Fanuc TP program (LS listing): HOME.LS

/PROG  HOME
/ATTR
OWNER		= MNEDITOR;
COMMENT		= "RobotSafePos";
PROG_SIZE	= 174;
CREATE		= DATE 26-08-17  TIME 11:20:48;
MODIFIED	= DATE 26-08-17  TIME 11:22:56;
FILE_NAME	= ;
VERSION		= 0;
LINE_COUNT	= 4;
MEMORY_SIZE	= 530;
PROTECT		= READ_WRITE;
TCD:  STACK_SIZE	= 0,
      TASK_PRIORITY	= 50,
      TIME_SLICE	= 0,
      BUSY_LAMP_OFF	= 0,
      ABORT_REQUEST	= 0,
      PAUSE_REQUEST	= 0;
DEFAULT_GROUP	= 1,*,*,*,*;
CONTROL_CODE	= 00000000 00000000;
LOCAL_REGISTERS	= 0,0,0;
/MN
   1:   ;
   2:   ;
   3:J PR[1:HOME_POSITION] 100% FINE    ;
   4:   ;
/POS
/END
